{attribute addProperty BoxType "EL6201-0000-0017"}
{attribute addProperty Id "Slave_14A_DI0BIT10.125105Slave_14A_DI1BIT10.125106Slave_14A_DI2BIT10.125107Slave_14A_DI3BIT10.125108Slave_14B_DI0BIT10.125109Slave_14B_DI1BIT10.125110Slave_14B_DI2BIT10.125111Slave_14B_DI3BIT10.125112"}
{attribute addProperty CRC "2889206870"}
{attribute addProperty SizeInBites "8"}
{attribute addProperty SizeInBytes "1"}
TYPE Slave_14_Inputs_AC35CC56 :
STRUCT
	{attribute addProperty Name "Slave_14A_DI0"}
	Slave_14A_DI0 : BIT;
	{attribute addProperty Name "Slave_14A_DI1"}
	Slave_14A_DI1 : BIT;
	{attribute addProperty Name "Slave_14A_DI2"}
	Slave_14A_DI2 : BIT;
	{attribute addProperty Name "Slave_14A_DI3"}
	Slave_14A_DI3 : BIT;
	{attribute addProperty Name "Slave_14B_DI0"}
	Slave_14B_DI0 : BIT;
	{attribute addProperty Name "Slave_14B_DI1"}
	Slave_14B_DI1 : BIT;
	{attribute addProperty Name "Slave_14B_DI2"}
	Slave_14B_DI2 : BIT;
	{attribute addProperty Name "Slave_14B_DI3"}
	Slave_14B_DI3 : BIT;
END_STRUCT
END_TYPE

(* stored: Version 1.2.0.0, ProductVersion 3.1.4024.9
   DUT Slave_14_Inputs_AC35CC56: Id {77d18ad1-ff66-4a04-b6c1-a9d397d81370} *)
